Yaskawa INFORM job: SKRZYNIA_4940_0_STOPNI_1OBR.JBI

/JOB
//NAME SKRZYNIA_4940_0_STOPNI_1OBR
///FOLDERNAME 02-SKRZYNIE_JOBS
//POS
///NPOS 518,518,0,43,0,0
///TOOL 0
///POSTYPE PULSE
///PULSE
C00000=1055,-24125,84372,288,19725,204
C00001=1055,-24125,84372,288,19725,204
C00002=0,-15438,65714,0,-68532,0
C00003=25524,-25821,36823,19654,-58495,38520
C00004=23988,-24960,37134,18595,-57837,38812
C00005=22822,-23954,37534,17811,-57199,39017
C00006=22935,-24057,37491,17887,-57262,38997
C00007=20006,-24258,37408,15644,-56932,39751
C00008=24402,-25289,37013,18874,-58060,38740
C00009=22585,-24665,40358,17164,-59622,30036
C00010=23477,-23257,40205,18030,-58646,29630
C00011=22519,-22398,40568,17384,-58125,29795
C00012=22700,-22567,40495,17506,-58225,29764
C00013=19339,-22794,40398,14955,-57865,30607
C00014=24825,-24328,39798,18931,-59350,29401
C00015=0,-15438,65714,0,-68532,0
C00016=25524,-25821,36823,19654,-58495,38520
C00017=23988,-24960,37134,18595,-57837,38812
C00018=22822,-23954,37534,17811,-57199,39017
C00019=22935,-24057,37491,17887,-57262,38997
C00020=20006,-24258,37408,15644,-56932,39751
C00021=24402,-25289,37013,18874,-58060,38740
C00022=22585,-24665,40358,17164,-59622,30036
C00023=23477,-23257,40205,18030,-58646,29630
C00024=22519,-22398,40568,17384,-58125,29795
C00025=22700,-22567,40495,17506,-58225,29764
C00026=19339,-22794,40398,14955,-57865,30607
C00027=24825,-24328,39798,18931,-59350,29401
C00028=32755,-32613,25711,29640,-48730,33694
C00029=25632,-30899,26166,23992,-46203,35378
C00030=24264,-29862,26497,22996,-45413,35639
C00031=24403,-29974,26459,23097,-45496,35612
C00032=20575,-30233,26374,19602,-44891,36810
C00033=26556,-31526,25988,24663,-46720,35206
C00034=30467,-34548,18624,42252,-31099,25545
C00035=27667,-31817,21023,40298,-29340,25942
C00036=26226,-30681,21430,39338,-28403,26129
C00037=26403,-30829,21375,39455,-28520,26106
C00038=23300,-31093,21277,35654,-27590,27434
C00039=27667,-31817,21023,40298,-29340,25942
C00040=26028,-43665,26580,-39946,8682,24640
C00041=27956,-30595,53065,-101898,6609,54413
C00042=26028,-43663,26580,-39944,8677,24639
C00043=38124,-35330,25507,26155,-45940,34419
C00044=17528,-33021,25719,14295,-44761,40001
C00045=28412,-21339,35361,20830,-70681,36412
C00046=27333,-20260,35973,20228,-70115,36596
C00047=27560,-20497,35837,20355,-70235,36556
C00048=24830,-20816,35654,18694,-69859,37222
C00049=28877,-18893,40191,20941,-72149,36569
C00050=27817,-32566,25782,25532,-47502,36865
C00051=25779,-31294,26110,24054,-46400,37243
C00052=24344,-30243,26427,23007,-45578,37515
C00053=24432,-30312,26405,23072,-45630,37498
C00054=20021,-30599,26315,19050,-44944,38872
C00055=26262,-31616,26021,24405,-46667,37153
C00056=27439,-32346,25835,25259,-47302,36935
C00057=25659,-31170,26146,23974,-46312,37260
C00058=24581,-30384,26384,23190,-45695,37464
C00059=24689,-30466,26358,23269,-45758,37444
C00060=20001,-30771,26264,18999,-45026,38899
C00061=26308,-31607,26026,24448,-46671,37139
C00062=29920,-29398,24569,49034,-27892,27689
C00063=29115,-28721,24834,48649,-27358,27707
C00064=27674,-27540,25333,47889,-26423,27783
C00065=27794,-27645,25287,47952,-26502,27777
C00066=24751,-27949,25156,44290,-25406,29014
C00067=29115,-28721,24834,48649,-27358,27707
C00068=46709,-36638,22429,58955,-37174,26391
C00069=28781,-29734,22128,31822,13650,18140
C00070=28781,-29734,22128,31822,47214,18140
C00071=28781,-29734,22128,31822,47214,18140
C00072=54276,-43673,-470,62120,-47739,23626
C00073=41752,-40945,238,55421,-40682,25053
C00074=39867,-39951,547,54583,-39468,25162
C00075=39963,-40004,529,54625,-39531,25157
C00076=37168,-40414,400,52318,-38319,25966
C00077=43368,-42081,-2849,57747,-40820,23950
C00078=38095,-40136,7813,41252,-44156,24924
C00079=33231,-38681,8176,37792,-41757,25918
C00080=31538,-37640,8473,36716,-40716,26179
C00081=31687,-37737,8444,36811,-40809,26155
C00082=27389,-38154,8322,32773,-39589,27627
C00083=33834,-39023,8084,38175,-42120,25821
C00084=27585,-47842,-289,32095,-40789,28095
C00085=4801,-35772,25187,4593,-28023,-82032
C00086=17634,-23800,39238,9573,-31425,-73339
C00087=17634,-23800,39238,9573,-31425,-73339
C00088=16549,-22464,39800,8390,-30730,-72975
C00089=16684,-22641,39722,8536,-30818,-73021
C00090=16684,-19968,45512,8078,-32771,-72767
C00091=17634,-23800,39238,9573,-31425,-73339
C00092=17837,-21535,44509,9322,-33342,-73155
C00093=17837,-21535,44509,9322,-33342,-73155
C00094=16866,-20378,45014,8305,-32755,-72853
C00095=17032,-20588,44918,8481,-32857,-72905
C00096=17032,-17542,51480,8009,-35060,-72636
C00097=17837,-21535,44509,9322,-33342,-73155
C00098=-20829,-18800,50532,-12466,-37179,-77446
C00099=-19934,-17904,50946,-11618,-36715,-77676
C00100=-20044,-18019,50891,-11723,-36773,-77647
C00101=-20044,-15288,56753,-11218,-38713,-77950
C00102=-20966,-18928,50473,-12596,-37250,-77413
C00103=-20884,-26676,33664,-14451,-31668,-76336
C00104=-20884,-26676,33664,-14451,-31668,-76336
C00105=-19557,-25338,34176,-13080,-30873,-76751
C00106=-19691,-25483,34117,-13220,-30955,-76709
C00107=-19691,-22773,39998,-12506,-32911,-77106
C00108=-20642,-26447,33747,-14206,-31526,-76411
C00109=-33629,-40566,17444,-29603,-33447,-71192
C00110=-33629,-40566,17444,42578,-32312,-84654
C00111=-42160,-31266,16400,42578,-32312,-84654
C00112=-87798,-804,48829,-20188,-26072,-60966
C00113=-76454,-11934,10236,-25964,7954,-64922
C00114=-76448,-11928,10235,-25961,7944,-64914
C00115=-68643,-7759,-23318,-14097,50582,-74897
C00116=-70868,-8793,-8075,-29663,30364,-70765
C00117=-67243,-1968,12282,-49553,26687,-63567
C00118=-68655,-309,14069,-48513,25966,-64203
C00119=-67497,-1678,12591,-49367,26558,-63682
C00120=-71436,-723,2905,-26484,35140,-73726
C00121=-71436,176,6426,-27636,33595,-73066
C00122=-71434,778,8668,-28412,32633,-72624
C00123=-68624,-2689,-85,-28291,36551,-72622
C00124=-99375,3692,5712,40719,48607,-84097
C00125=-94964,4957,10918,40408,44640,-83792
C00126=-93063,6047,12199,39572,43744,-83178
C00127=-94964,4957,10918,40408,44640,-83792
C00128=-94964,5754,13918,41385,43553,-84439
C00129=-94964,4957,10918,40408,44640,-83792
C00130=-90271,-412,-5146,23417,46876,-76529
C00131=-83133,-4088,-8267,6704,41492,-71542
C00132=-83133,-4088,-8267,6704,41492,-71542
C00133=-83133,-4088,-8267,6704,41492,-11598
C00134=-83133,-16026,-8267,6704,41492,-11598
C00135=-83133,-16026,-8267,6704,41492,-11598
C00136=-48225,-19387,30619,3889,32460,-6728
C00137=56943,-39861,25115,1795,-37402,-69601
C00138=29960,-38386,-19607,-115769,-41858,-24264
C00139=65721,-6478,18155,-133323,-22195,3361
C00140=70544,4411,32968,-134868,-18623,4660
C00141=71874,8263,38598,-134556,-17327,4659
C00142=72629,9390,40002,-135279,-16924,5107
C00143=71441,7638,37831,-134139,-17555,4406
C00144=77146,8888,25050,-166574,-32612,18372
C00145=77146,10029,28643,-166204,-31014,18167
C00146=77146,11198,32202,-165803,-29459,17947
C00147=75508,4678,16951,-165715,-35157,17778
C00148=68680,12216,24468,-164340,-40455,-13359
C00149=68362,12845,25743,-164045,-40097,-13561
C00150=68362,13700,28585,-163752,-38808,-13742
C00151=68362,12845,25743,-164045,-40097,-13561
C00152=64993,-1168,28876,-102971,-10760,-49875
C00153=63888,481,30670,-102324,-11438,-50313
C00154=64993,-1168,28876,-102971,-10760,-49875
C00155=58588,-14653,4620,-120782,-19611,-35794
C00156=29960,-38386,-19607,-115769,-41858,-24264
C00157=56943,-39861,25115,1795,-37402,-69601
C00158=-1002,-39861,25115,1795,-37402,-69601
C00159=-1001,-39858,25114,1795,-37402,0
C00160=6591,-33902,35532,5956,-1761,-1932
C00161=6592,-33900,35531,103508,-35512,-26314
C00162=-99253,-13690,44082,59847,13407,-31313
C00163=-85045,-36869,-4353,28502,-22832,-52282
C00164=-92346,-18713,13565,21110,-22545,-55257
C00165=-85732,-21202,11427,30682,-24763,-59235
C00166=-84559,-15616,15722,33768,-24118,-60665
C00167=-84150,-13282,17685,34842,-23935,-61163
C00168=-83260,-12880,18034,36130,-24218,-61709
C00169=-84150,-13282,17685,34842,-23935,-61163
C00170=-85365,-11775,19006,33430,-23307,-60600
C00171=-84150,-13282,17685,34842,-23935,-61163
C00172=-85786,-16909,14677,31743,-23900,-59790
C00173=-84150,-13282,17685,34842,-23935,-61163
C00174=-83215,-12861,18051,36194,-24233,-61735
C00175=-84150,-13282,17685,34842,-23935,-61163
C00176=-85327,-11825,18959,33476,-23327,-60618
C00177=-84150,-13282,17685,34842,-23935,-61163
C00178=-87841,-18519,13420,28367,-23534,-58339
C00179=-84150,-13282,17685,34842,-23935,-61163
C00180=-83292,-12894,18020,36083,-24208,-61688
C00181=-84150,-13282,17685,34842,-23935,-61163
C00182=-85185,-12008,18799,33646,-23400,-60687
C00183=-84150,-13282,17685,34842,-23935,-61163
C00184=-86371,-18277,13606,30568,-23951,-59265
C00185=-84345,-13370,17612,34554,-23873,-61041
C00186=-83240,-12871,18042,36158,-24225,-61720
C00187=-84345,-13370,17612,34554,-23873,-61041
C00188=-85365,-12110,18711,33368,-23345,-60568
C00189=-84345,-13370,17612,34554,-23873,-61041
C00190=-86191,-19647,12567,30467,-24278,-59187
C00191=-84345,-13372,17610,34552,-23873,-61039
C00192=-83096,-12807,18098,36363,-24268,-61804
C00193=-84345,-13372,17610,34552,-23873,-61039
C00194=-85268,-12232,18600,33480,-23393,-60612
C00195=-84345,-13372,17610,34552,-23873,-61039
C00196=-84814,-16043,15376,33312,-24093,-60464
C00197=-84104,-13265,17702,34906,-23948,-61189
C00198=-82960,-12743,18153,36555,-24313,-61887
C00199=-84104,-13265,17702,34906,-23948,-61189
C00200=-84979,-12194,18635,33901,-23496,-60788
C00201=-84104,-13265,17702,34906,-23948,-61189
C00202=-86610,-16845,14732,30573,-23614,-59301
C00203=-84104,-13265,17702,34906,-23948,-61189
C00204=-82793,-12667,18222,36790,-24370,-61986
C00205=-84104,-13265,17702,34906,-23948,-61189
C00206=-84888,-12305,18537,34004,-23540,-60830
C00207=-84104,-13265,17702,34906,-23948,-61189
C00208=-83806,-19585,12613,33764,-25080,-60559
C00209=-83675,-13072,17868,35530,-24083,-61453
C00210=-82553,-12556,18319,37130,-24451,-62127
C00211=-83675,-13072,17868,35530,-24083,-61453
C00212=-84378,-12223,18610,34735,-23716,-61138
C00213=-83675,-13072,17868,35530,-24083,-61453
C00214=-87149,-17993,13826,29513,-23647,-58830
C00215=-84104,-13265,17702,34906,-23948,-61189
C00216=-82640,-12594,18285,37014,-24425,-62079
C00217=-84104,-13265,17702,34906,-23948,-61189
C00218=-84792,-12429,18430,34119,-23592,-60877
C00219=-84104,-13265,17702,34906,-23948,-61189
C00220=-83583,-9185,30892,23668,-36042,-57025
C00221=-85789,-8328,35795,20592,-37093,-55378
C00222=-85786,-16735,14816,31782,-23869,-59812
C00223=-84103,-13263,17702,34906,-23947,-61191
C00224=-83225,-12865,18046,36177,-24227,-61729
C00225=-84103,-13263,17702,34906,-23947,-61191
C00226=-84774,-12447,18412,34138,-23599,-60886
C00227=-84103,-13263,17702,34906,-23947,-61191
C00228=-86149,-16246,6730,18897,-35239,-57128
C00229=-86244,-15289,7532,18875,-35060,-57127
C00230=-85361,-14893,7870,19824,-35193,-57574
C00231=-86244,-15289,7532,18875,-35060,-57127
C00232=-86889,-14409,8282,18264,-34784,-56850
C00233=-86244,-15289,7532,18875,-35060,-57127
C00234=-90262,-21765,2389,14114,-35574,-54847
C00235=-90262,-21765,2389,28730,-17672,-54847
C00236=-89967,-19086,25635,28730,-17672,-54847
C00237=568,-24029,84339,168,19981,112
C00238=568,-24677,83015,164,20405,113
C00239=101153,-24598,83176,165,20353,113
C00240=101153,-24598,83176,165,20353,113
C00241=89967,-19086,25635,-28730,-17672,54847
C00242=90262,-21765,2389,-28730,-17672,54847
C00243=86932,-18662,4771,-17876,-35519,56628
C00244=86578,-15436,7408,-18515,-35011,56957
C00245=85428,-14922,7844,-19753,-35183,57541
C00246=84405,-14447,8250,-20842,-35348,58054
C00247=85428,-14922,7844,-19753,-35183,57541
C00248=86134,-13973,8661,-19091,-34881,57237
C00249=85428,-14922,7844,-19753,-35183,57541
C00250=85786,-16735,14816,-31782,-23869,59812
C00251=83514,-12996,17929,-35760,-24132,61552
C00252=82296,-12429,18424,-37488,-24534,62281
C00253=83514,-12996,17929,-35760,-24132,61552
C00254=84266,-12085,18725,-34910,-23738,61214
C00255=83514,-12996,17929,-35760,-24132,61552
C00256=87323,-6914,39851,-18853,-38149,44508
C00257=83118,-12818,18089,-36330,-24263,61791
C00258=81969,-12276,18566,-37944,-24648,62472
C00259=83118,-12818,18089,-36330,-24263,61791
C00260=83927,-11846,18941,-35423,-23842,61433
C00261=83118,-12818,18089,-36330,-24263,61791
C00262=83806,-19585,12613,-33764,-25080,60559
C00263=83148,-12832,18077,-36287,-24254,61773
C00264=81889,-12236,18598,-38058,-24676,62520
C00265=83148,-12832,18077,-36287,-24254,61773
C00266=83900,-11930,18867,-35446,-23862,61440
C00267=83148,-12832,18077,-36287,-24254,61773
C00268=86610,-16845,14732,-30573,-23614,59301
C00269=82493,-13239,17725,-37070,-24559,62089
C00270=81442,-12739,18159,-38529,-24915,62703
C00271=82493,-13239,17725,-37070,-24559,62089
C00272=83435,-12133,18689,-36040,-24063,61682
C00273=82493,-13239,17725,-37070,-24559,62089
C00274=84814,-16043,15376,-33312,-24093,60464
C00275=82555,-13613,17404,-36910,-24580,62015
C00276=81369,-13053,17885,-38558,-24979,62709
C00277=82555,-13613,17404,-36910,-24580,62015
C00278=83568,-12431,18429,-35805,-24046,61580
C00279=82555,-13613,17404,-36910,-24580,62015
C00280=86191,-19647,12567,-30467,-24278,59187
C00281=82500,-13648,17375,-36975,-24607,62039
C00282=81594,-13224,17740,-38236,-24911,62571
C00283=82500,-13648,17375,-36975,-24607,62039
C00284=83449,-12543,18332,-35941,-24104,61633
C00285=82500,-13648,17375,-36975,-24607,62039
C00286=86371,-18277,13606,-30568,-23951,59265
C00287=82904,-13790,17251,-36416,-24470,61808
C00288=81796,-13275,17692,-37971,-24838,62464
C00289=82904,-13790,17251,-36416,-24470,61808
C00290=83696,-12867,18046,-35547,-24051,61466
C00291=82904,-13790,17251,-36416,-24470,61808
C00292=87841,-18519,13420,-28367,-23534,58339
C00293=82748,-13879,17174,-36603,-24542,61883
C00294=81789,-13434,17554,-37946,-24861,62449
C00295=82748,-13879,17174,-36603,-24542,61883
C00296=83603,-12888,18026,-35668,-24086,61514
C00297=82748,-13879,17174,-36603,-24542,61883
C00298=85786,-16909,14677,-31743,-23900,59790
C00299=82339,-14116,16972,-37087,-24733,62079
C00300=81557,-13752,17280,-38171,-24994,62536
C00301=82339,-14116,16972,-37087,-24733,62079
C00302=83390,-12909,18006,-35951,-24172,61633
C00303=82339,-14116,16972,-37087,-24733,62079
C00304=85732,-21202,11427,-30682,-24763,59235
C00305=82398,-14365,16763,-36952,-24745,62014
C00306=81340,-13876,17176,-38416,-25096,62632
C00307=82398,-14365,16763,-36952,-24745,62014
C00308=83629,-12951,17972,-35620,-24090,61491
C00309=82398,-14365,16763,-36952,-24745,62014
C00310=83775,-36460,5778,-32556,-23750,56951
C00311=69856,-53931,-13446,-33557,-28911,29591
C00312=0,-24029,84339,0,19981,0
C00313=0,-24029,84339,0,19981,0
C00314=0,-52280,40443,0,6876,0
C00315=43695,-41610,22646,45477,-37580,9181
C00316=79833,-32060,29151,65065,-75499,17030
C00317=46589,-23543,32575,47437,-59456,19719
C00318=34746,-28644,20980,31794,-60034,26371
C00319=20694,-31959,9398,15734,-60691,34314
C00320=58029,-25484,23838,55879,-68285,17494
C00321=64424,-28491,31029,58630,-66351,17656
C00322=0,-52280,40443,0,6876,0
C00323=0,-52280,40443,0,6876,0
C00324=23755,-47704,18289,26329,-25233,13971
C00325=32804,-46073,6525,41905,-31120,14425
C00326=62562,-39100,6547,70046,-55853,12125
C00327=48126,-33841,8393,64372,-47199,12361
C00328=31253,-44096,-7366,36514,-42480,22085
C00329=59828,-44646,-5405,72855,-48572,12139
C00330=0,-38761,66314,0,-763,0
C00331=0,-44757,54667,0,2744,0
C00332=40382,-38226,12225,48505,-40693,16039
C00333=55481,-27484,23768,62968,-54833,11978
C00334=49931,-26522,24223,59987,-51967,12537
C00335=41382,-34078,10932,46059,-50502,16311
C00336=55330,-33748,11238,57660,-59334,12681
C00337=78664,-24436,10378,82837,-79111,12029
C00338=75189,-23065,11287,81851,-76948,11927
C00339=75189,-45249,11287,81851,-38847,11927
C00340=29880,-45249,11287,43145,-11324,11927
C00341=0,-24029,84339,0,19981,0
C00342=0,-24026,84338,1,19977,2
C00343=4264,-34194,25387,4006,-26954,-29436
C00344=4264,-34194,25387,4006,-26954,-81856
C00345=-21478,-27798,32214,-15234,-31599,-76056
C00346=-19679,-23059,39354,-12567,-32689,-77067
C00347=16724,-20576,44291,8212,-32395,-72836
C00348=21329,-26386,39716,13285,-34016,-74401
C00349=-23778,-26243,38799,-16502,-35132,-75964
C00350=-20075,-15782,55752,-11329,-38404,-77896
C00351=16874,-17447,51356,7863,-34895,-72604
C00352=18580,-28601,30698,11472,-29284,-74138
C00353=6126,-41331,18955,6697,-26557,-30383
C00354=1,-24024,84337,2,19973,1
C00355=-64243,-26178,31107,-39513,40312,-5844
C00356=-72148,3973,56008,-35470,42045,-10522
C00357=-72090,16396,76301,-42067,35650,-6519
C00358=-69388,15725,61378,-31740,35177,-8719
C00359=-69127,27099,75569,-32744,34250,-8088
C00360=-67573,2495,11285,-21767,57629,-15193
C00361=-77819,19629,29798,-10454,63174,-20704
C00362=-72990,23583,14304,-10735,77209,-20379
C00363=-74593,38003,46707,-11043,65751,-19814
C00364=-73236,38943,48295,-11400,65557,-19316
C00365=-73329,42107,51779,-6346,67443,-19636
C00366=-87142,34654,46174,17622,63862,-25393
C00367=-87240,36727,48611,18897,66604,-25032
C00368=-99033,21517,12213,24947,79702,-26203
C00369=-91500,-14196,-34781,24472,81625,-22832
C00370=-100472,-45007,-27818,8167,67201,-29302
C00371=0,-36642,16905,0,48372,0
C00372=66009,-61997,-62105,21406,63483,18379
C00373=97242,-23579,-39442,10179,68876,30321
C00374=73684,-7073,-17511,24638,68131,29022
C00375=59136,7235,6676,33270,66602,27507
C00376=54816,14937,6234,39741,69494,31070
C00377=54365,20668,19279,41017,66202,29418
C00378=64503,4223,2857,29650,48528,26647
C00379=75622,3202,-3149,3890,49494,34281
C00380=88036,13177,2413,-18568,66573,35876
C00381=90462,21593,10123,-22613,76266,34479
C00382=92450,29224,20002,-25750,81642,33727
C00383=94949,8131,-12163,-20291,74229,36861
C00384=94949,8084,-13484,-20215,75047,36712
C00385=70412,-34016,-52305,-11724,65624,29757
C00386=44268,-30306,-1568,-7370,48673,18708
C00387=1,-24024,84337,2,19973,1
C00388=1,-24024,84337,2,19973,1
C00389=3796,-57671,22373,2336,-25309,-753
C00390=52632,-34554,16626,51161,-63050,5622
C00391=41454,-25301,37199,36495,-58855,24340
C00392=36675,-26014,30916,36565,-54296,30358
C00393=31298,-42259,-4306,53964,-29254,17939
C00394=62932,-33588,12189,66848,-61063,18031
C00395=57521,-31202,17284,65112,-55174,10876
C00396=49869,-26949,23557,59706,-52171,12606
C00397=49645,-31441,12217,55064,-56016,13120
C00398=55330,-33748,11238,57660,-59334,12681
C00399=29694,-28537,50295,31543,-18263,8508
C00400=1,-24024,84337,2,19973,1
C00401=1,-24024,84337,2,19973,1
C00402=57188,-41777,19973,48132,-58706,4905
C00403=55566,-48748,-16991,79805,-45048,-6941
C00404=49908,-48716,-25784,90749,-41340,-3650
C00405=34097,-50090,-26426,85195,-27377,-3312
C00406=29342,-53468,-37504,108423,-23986,-15312
C00407=55456,-69347,-61742,105381,-46819,-11205
C00408=12119,-24859,71505,13236,4440,2633
C00409=-91085,-34291,10385,1908,-24348,-42097
C00410=-86191,-19647,12567,30467,-24278,-59187
C00411=-99336,-11722,19052,-14323,-20229,-40037
C00412=-98356,-11562,19564,-10422,-20330,-41507
C00413=-99474,-20389,12397,-11593,-22150,-41069
C00414=0,-52280,40443,0,6876,0
C00415=98750,-34911,19055,13387,-20552,33529
C00416=85481,-22689,10385,-30594,-25183,59147
C00417=97204,-12655,18233,8807,-19987,42423
C00418=97248,-12883,18033,8874,-20029,42393
C00419=96230,-24528,9149,6144,-22576,43630
C00420=0,-52280,40443,0,6876,0
C00421=0,-52280,40443,0,6876,0
C00422=-90140,-60305,18108,-2708,1721,-7625
C00423=-95594,-27428,6866,-4663,-19832,-42154
C00424=-99356,-13410,18355,-15385,-17730,-37479
C00425=-99591,-10931,20459,-16242,-17374,-37088
C00426=-99412,-10883,20509,-15863,-17339,-37249
C00427=-100555,-16348,15834,-17428,-18409,-36628
C00428=-90140,-60305,18108,-2708,1721,-7625
C00429=0,-52280,40443,0,6876,0
C00430=84259,-57935,27522,-3761,3673,6310
C00431=86507,-39672,4297,-27618,-16640,46340
C00432=79502,-31038,5321,-35142,-29552,60614
C00433=87509,-17632,14108,-29072,-23467,58651
C00434=100494,-12641,18246,19637,-20925,37756
C00435=99867,-15453,10402,24266,-14765,33998
C00436=100699,-20865,6123,24471,-16015,33991
C00437=86507,-39672,4297,-27618,-16640,46340
C00438=84259,-57935,27522,-3761,3673,6310
C00439=0,-52280,40443,0,6876,0
C00440=0,-27933,77061,0,20812,0
C00441=0,-27933,77061,0,20812,0
C00442=0,-52280,40443,0,6876,0
C00443=-91970,-60791,14435,-3343,512,-9412
C00444=-99196,-15868,16098,-13748,-19297,-38710
C00445=-99196,-15868,16098,-13748,-19297,-38710
C00446=-99196,-15868,16098,-13748,-19297,-38710
C00447=-85896,-11794,19566,31613,-21074,-58206
C00448=-87494,-11929,19445,26784,-20178,-56163
C00449=-99562,-16264,15781,-14410,-19427,-38431
C00450=-99196,-15868,16098,-13748,-19297,-38710
C00451=-91970,-60791,14435,-3343,512,-9412
C00452=0,-52280,40443,0,6876,0
C00453=91083,-60784,14823,-9043,-825,15173
C00454=83869,-19403,12921,-33769,-24740,60260
C00455=83869,-19403,12921,-33769,-24740,60260
C00456=83420,-14897,16486,-35538,-24144,61113
C00457=90681,-11839,19658,-13770,-20778,51433
C00458=90505,-11641,19895,-14005,-20849,51502
C00459=95871,-14889,15992,4901,-19605,43825
C00460=83869,-19403,12921,-33769,-24740,60260
C00461=91083,-60784,14823,-9043,-825,15173
C00462=0,-52280,40443,0,6876,0
C00463=-91526,-60598,16699,7584,176,-13289
C00464=-94392,-6553,48683,5805,-47321,-49764
C00465=-88951,-345,54953,10686,-47392,-51569
C00466=-88305,5764,62037,11205,-47732,-51744
C00467=-91201,-14114,9416,8552,-34389,-51801
C00468=-84917,-15593,15742,33275,-23984,-60461
C00469=-81669,-15982,15425,37506,-25258,-62202
C00470=-79867,-25377,9541,37586,-25936,-59971
C00471=-91415,-60262,16631,7870,-73,-13734
C00472=24,-24029,84339,7,19981,5
C00473=160,-24029,84339,47,19981,32
C00474=99096,-24029,84339,47,19981,32
C00475=99096,-24029,84339,47,19981,32
C00476=89967,-19086,25635,-28730,-17672,54847
C00477=85786,-16735,14816,-31782,-23869,59812
C00478=83492,-14473,16674,-35480,-24338,61406
C00479=82747,-11488,19289,-37317,-24361,62210
C00480=85506,-13730,8787,-19466,-34817,57474
C00481=85505,-16299,6686,-19564,-35388,57437
C00482=89967,-19086,25635,-28730,-17672,54847
C00483=568,-24029,84339,168,19981,112
C00484=568,-24029,84339,168,19981,112
C00485=-91970,-60791,14435,-3343,512,-9412
C00486=-86948,-23217,10819,28314,-23349,-56438
C00487=-85895,-16522,15767,31843,-22281,-58087
C00488=-93744,1669,52928,2829,-38206,-34736
C00489=-93484,-766,47198,3260,-36104,-34933
C00490=-86145,-24679,9854,29028,-23971,-56682
C00491=-100471,-58311,4157,14142,-4822,-27614
C00492=-68517,-58311,4157,14142,-4822,-27614
C00493=0,-52280,40443,0,6876,0
C00494=91083,-60784,14823,-9043,-825,15173
C00495=83869,-19403,12921,-33769,-24740,60260
C00496=82620,-18743,14708,-32942,-26226,58979
C00497=84031,-4887,35984,-19530,-40379,54984
C00498=84316,-7987,27276,-19995,-38113,55712
C00499=84798,-22668,11879,-29033,-26372,57255
C00500=91083,-60784,14823,-9043,-825,15173
C00501=0,-52280,40443,0,6876,0
C00502=-6369,-39206,65423,-4801,-482,2563
C00503=-97287,-29142,12714,-8673,-22288,-37832
C00504=-86191,-19647,12567,30467,-24278,-59187
C00505=-85671,-16302,15857,30808,-24404,-58999
C00506=-100216,-10426,22391,-15020,-22581,-38655
C00507=-96259,-10424,22189,-2878,-17380,-43087
C00508=-87910,-17792,15835,25414,-24996,-56048
C00509=-97287,-29142,12714,-8673,-22288,-37832
C00510=0,-52280,40443,0,6876,0
C00511=92301,-25634,22749,2368,-15645,37646
C00512=83738,-18329,13570,-34202,-24868,60772
C00513=90255,-12942,18284,-15153,-20833,52586
C00514=93508,-13158,18002,-4292,-20124,47959
C00515=80226,-20465,12178,-39626,-27411,62762
C00516=92301,-25634,22749,2368,-15645,37646
C00517=0,-52280,40443,0,6876,0
BC00000=413138
BC00001=413138
BC00002=413138
BC00003=290246
BC00004=290246
BC00005=290246
BC00006=290246
BC00007=290246
BC00008=290246
BC00009=347127
BC00010=347132
BC00011=347132
BC00012=347132
BC00013=347132
BC00014=347132
BC00015=413138
BC00016=413134
BC00017=413134
BC00018=413134
BC00019=413134
BC00020=413134
BC00021=413134
BC00022=474623
BC00023=474628
BC00024=474628
BC00025=474628
BC00026=474628
BC00027=474628
BC00028=522849
BC00029=522849
BC00030=522849
BC00031=522849
BC00032=522849
BC00033=522849
BC00034=550624
BC00035=553627
BC00036=553627
BC00037=553627
BC00038=553627
BC00039=553627
BC00040=470246
BC00041=618860
BC00042=673957
BC00043=691345
BC00044=686969
BC00045=712250
BC00046=712250
BC00047=712250
BC00048=712250
BC00049=712250
BC00050=708270
BC00051=708270
BC00052=708270
BC00053=708270
BC00054=708270
BC00055=708270
BC00056=770184
BC00057=770184
BC00058=770184
BC00059=770184
BC00060=770184
BC00061=770184
BC00062=788736
BC00063=788736
BC00064=788736
BC00065=788736
BC00066=788736
BC00067=788736
BC00068=729895
BC00069=703565
BC00070=703565
BC00071=802913
BC00072=891475
BC00073=891475
BC00074=891475
BC00075=891475
BC00076=891475
BC00077=891475
BC00078=934475
BC00079=934475
BC00080=934475
BC00081=934475
BC00082=934475
BC00083=934475
BC00084=934475
BC00085=880430
BC00086=895791
BC00087=895791
BC00088=895791
BC00089=895791
BC00090=895791
BC00091=895791
BC00092=900237
BC00093=900237
BC00094=900237
BC00095=900237
BC00096=900237
BC00097=900237
BC00098=900237
BC00099=900237
BC00100=900237
BC00101=900237
BC00102=900237
BC00103=900237
BC00104=900237
BC00105=900237
BC00106=900237
BC00107=900237
BC00108=900237
BC00109=900237
BC00110=900237
BC00111=900237
BC00112=900237
BC00113=900237
BC00114=917989
BC00115=929075
BC00116=945779
BC00117=945779
BC00118=945779
BC00119=945779
BC00120=945779
BC00121=945779
BC00122=945780
BC00123=945780
BC00124=945780
BC00125=945780
BC00126=945780
BC00127=945780
BC00128=945780
BC00129=945780
BC00130=936157
BC00131=921523
BC00132=896258
BC00133=896258
BC00134=896258
BC00135=863076
BC00136=828643
BC00137=900237
BC00138=900237
BC00139=900237
BC00140=916451
BC00141=921612
BC00142=921612
BC00143=921612
BC00144=921612
BC00145=921612
BC00146=921612
BC00147=921612
BC00148=921612
BC00149=921612
BC00150=921612
BC00151=921612
BC00152=921612
BC00153=921612
BC00154=921612
BC00155=916099
BC00156=869515
BC00157=838793
BC00158=838793
BC00159=854156
BC00160=785093
BC00161=785096
BC00162=785096
BC00163=854699
BC00164=886829
BC00165=902188
BC00166=902188
BC00167=902188
BC00168=902188
BC00169=902188
BC00170=902188
BC00171=902188
BC00172=840744
BC00173=840744
BC00174=840744
BC00175=840744
BC00176=840744
BC00177=840744
BC00178=779300
BC00179=779300
BC00180=779300
BC00181=779300
BC00182=779300
BC00183=779300
BC00184=717855
BC00185=717855
BC00186=717855
BC00187=717855
BC00188=717855
BC00189=717855
BC00190=656405
BC00191=656405
BC00192=656405
BC00193=656405
BC00194=656405
BC00195=656405
BC00196=594961
BC00197=594961
BC00198=594961
BC00199=594961
BC00200=594961
BC00201=594961
BC00202=533517
BC00203=533517
BC00204=533517
BC00205=533517
BC00206=533517
BC00207=533517
BC00208=472073
BC00209=472073
BC00210=472073
BC00211=472073
BC00212=472073
BC00213=472073
BC00214=410629
BC00215=410629
BC00216=410629
BC00217=410629
BC00218=410629
BC00219=410629
BC00220=410629
BC00221=349186
BC00222=349186
BC00223=349186
BC00224=349186
BC00225=349186
BC00226=349186
BC00227=349186
BC00228=336469
BC00229=336469
BC00230=336469
BC00231=336469
BC00232=336469
BC00233=336469
BC00234=336469
BC00235=336469
BC00236=336469
BC00237=336469
BC00238=511557
BC00239=512005
BC00240=363797
BC00241=336469
BC00242=336469
BC00243=337415
BC00244=337415
BC00245=337415
BC00246=337415
BC00247=337415
BC00248=337415
BC00249=337415
BC00250=349186
BC00251=350137
BC00252=350137
BC00253=350137
BC00254=350137
BC00255=350137
BC00256=410629
BC00257=411580
BC00258=411580
BC00259=411580
BC00260=411580
BC00261=411580
BC00262=472073
BC00263=473025
BC00264=473025
BC00265=473025
BC00266=473025
BC00267=473025
BC00268=533517
BC00269=534468
BC00270=534468
BC00271=534468
BC00272=534468
BC00273=534468
BC00274=594961
BC00275=594961
BC00276=594961
BC00277=594961
BC00278=594961
BC00279=594961
BC00280=656405
BC00281=657350
BC00282=657350
BC00283=657350
BC00284=657350
BC00285=657350
BC00286=717855
BC00287=718799
BC00288=718799
BC00289=718799
BC00290=718799
BC00291=718799
BC00292=779300
BC00293=780245
BC00294=780245
BC00295=780245
BC00296=780245
BC00297=780245
BC00298=840744
BC00299=841691
BC00300=841691
BC00301=841691
BC00302=841691
BC00303=841691
BC00304=902188
BC00305=903136
BC00306=903136
BC00307=903136
BC00308=903136
BC00309=903136
BC00310=866428
BC00311=742376
BC00312=673191
BC00313=769966
BC00314=716865
BC00315=723595
BC00316=717171
BC00317=717171
BC00318=716481
BC00319=715784
BC00320=716000
BC00321=727625
BC00322=716865
BC00323=820009
BC00324=882789
BC00325=908954
BC00326=917484
BC00327=934308
BC00328=923719
BC00329=887066
BC00330=801718
BC00331=499733
BC00332=475338
BC00333=456696
BC00334=456696
BC00335=417276
BC00336=417276
BC00337=493986
BC00338=514306
BC00339=485368
BC00340=478024
BC00341=473587
BC00342=774064
BC00343=862181
BC00344=867397
BC00345=900237
BC00346=900237
BC00347=895790
BC00348=890024
BC00349=885535
BC00350=900237
BC00351=900237
BC00352=899465
BC00353=903057
BC00354=750918
BC00355=766280
BC00356=766280
BC00357=822990
BC00358=842876
BC00359=867815
BC00360=899747
BC00361=899747
BC00362=927256
BC00363=927256
BC00364=927256
BC00365=927257
BC00366=927257
BC00367=927258
BC00368=927258
BC00369=927258
BC00370=841916
BC00371=800514
BC00372=884054
BC00373=923174
BC00374=923175
BC00375=923175
BC00376=953422
BC00377=953422
BC00378=953422
BC00379=953422
BC00380=953422
BC00381=953425
BC00382=953425
BC00383=953425
BC00384=927019
BC00385=927019
BC00386=858206
BC00387=735557
BC00388=469153
BC00389=499904
BC00390=541592
BC00391=531564
BC00392=529848
BC00393=579756
BC00394=529848
BC00395=333808
BC00396=332068
BC00397=295166
BC00398=294388
BC00399=454783
BC00400=441730
BC00401=632615
BC00402=778314
BC00403=778312
BC00404=778312
BC00405=778312
BC00406=835726
BC00407=836556
BC00408=566410
BC00409=707357
BC00410=656405
BC00411=656405
BC00412=717855
BC00413=717855
BC00414=680147
BC00415=662303
BC00416=657350
BC00417=657350
BC00418=718803
BC00419=718803
BC00420=683493
BC00421=792672
BC00422=792672
BC00423=896850
BC00424=895720
BC00425=895720
BC00426=925351
BC00427=927080
BC00428=792672
BC00429=792672
BC00430=792672
BC00431=887446
BC00432=903126
BC00433=903126
BC00434=903126
BC00435=936389
BC00436=936389
BC00437=887446
BC00438=792672
BC00439=792672
BC00440=700249
BC00441=546214
BC00442=546214
BC00443=546211
BC00444=546211
BC00445=406776
BC00446=406776
BC00447=406778
BC00448=468200
BC00449=468200
BC00450=546211
BC00451=546211
BC00452=546214
BC00453=546214
BC00454=507604
BC00455=410782
BC00456=410782
BC00457=410782
BC00458=472720
BC00459=472720
BC00460=507604
BC00461=546214
BC00462=546214
BC00463=516757
BC00464=383716
BC00465=349186
BC00466=349186
BC00467=336469
BC00468=349186
BC00469=410629
BC00470=416512
BC00471=515801
BC00472=520018
BC00473=474013
BC00474=474013
BC00475=403108
BC00476=336469
BC00477=349186
BC00478=349186
BC00479=349186
BC00480=337415
BC00481=337415
BC00482=336469
BC00483=336469
BC00484=428401
BC00485=546211
BC00486=591088
BC00487=591088
BC00488=591088
BC00489=531116
BC00490=529640
BC00491=529640
BC00492=529640
BC00493=529640
BC00494=546214
BC00495=589919
BC00496=595627
BC00497=609761
BC00498=555903
BC00499=534177
BC00500=546214
BC00501=529640
BC00502=651195
BC00503=765890
BC00504=777968
BC00505=778453
BC00506=779252
BC00507=832733
BC00508=840748
BC00509=730002
BC00510=671551
BC00511=714120
BC00512=780224
BC00513=780222
BC00514=841743
BC00515=841743
BC00516=741100
BC00517=660586
///POSTYPE BASE
///RECTAN
///RCONF 1,0,0,0,0,0,0,0,0,0,0,0,0,0,0,0,0,0,0,0,0,0,0,0
P00006=0.000,0.000,0.000,0.0000,0.0000,0.0000
///RCONF 0,0,0,0,0,0,0,0,0,0,0,0,0,0,0,0,0,0,0,0,0,0,0,0
P00021=6.550,-0.003,-5.735,0.0000,0.0000,0.0000
P00022=5.943,-0.018,-6.388,0.0000,0.0000,0.0000
P00023=7.025,-0.019,-7.168,0.0000,0.0000,0.0000
P00024=5.926,-0.047,-4.777,0.0000,0.0000,0.0000
///RCONF 1,0,0,0,0,0,0,0,0,0,0,0,0,0,0,0,0,0,0,0,0,0,0,0
P00098=-0.089,-2.467,4.059,0.0000,0.0000,0.0000
P00099=0.011,-2.380,1.226,0.0000,0.0000,0.0000
P00100=-0.081,2.558,4.482,0.0000,0.0000,0.0000
P00101=0.030,-2.286,2.993,0.0000,0.0000,0.0000
P00102=-0.005,-1.108,1.644,0.0000,0.0000,0.0000
P00103=-0.094,-3.400,4.200,0.0000,0.0000,0.0000
P00104=0.043,-2.127,5.826,0.0000,0.0000,0.0000
P00105=-0.043,0.662,5.286,0.0000,0.0000,0.0000
P00106=-0.018,-2.519,0.237,0.0000,0.0000,0.0000
P00107=-0.008,-4.537,-4.500,0.0000,0.0000,0.0000
P00108=0.014,-3.040,2.637,0.0000,0.0000,0.0000
P00109=0.017,-3.622,2.341,0.0000,0.0000,0.0000
///RCONF 0,0,0,0,0,0,0,0,0,0,0,0,0,0,0,0,0,0,0,0,0,0,0,0
P00280=-0.761,-1.221,0.004,0.0000,0.0000,0.0000
///RCONF 1,0,0,0,0,0,0,0,0,0,0,0,0,0,0,0,0,0,0,0,0,0,0,0
P00281=-0.866,-3.587,-0.008,0.0000,0.0000,0.0000
///RCONF 0,0,0,0,1,0,0,0,0,0,0,0,0,0,0,0,0,0,0,0,0,0,0,0
P00290=-0.023,-0.050,5.560,0.0000,0.0000,0.0000
///RCONF 1,0,0,0,0,0,0,0,0,0,0,0,0,0,0,0,0,0,0,0,0,0,0,0
P00291=0.002,-0.893,4.526,0.0000,0.0000,0.0000
P00301=0.046,-2.112,7.779,0.0000,0.0000,0.0000
P00302=-0.180,-2.409,6.326,0.0000,0.0000,0.0000
///RCONF 0,0,0,0,0,0,0,0,0,0,0,0,0,0,0,0,0,0,0,0,0,0,0,0
P00303=-0.004,-1.437,-4.584,0.0000,0.0000,0.0000
P00304=0.028,-1.666,-4.234,0.0000,0.0000,0.0000
P00305=-0.003,-1.920,-3.501,0.0000,0.0000,0.0000
P00306=0.015,-2.252,-3.054,0.0000,0.0000,0.0000
P00307=0.019,-2.151,-5.077,0.0000,0.0000,0.0000
P00308=-0.003,-2.092,-4.888,0.0000,0.0000,0.0000
P00309=-0.040,-2.205,-4.992,0.0000,0.0000,0.0000
P00310=-0.006,-2.490,-5.925,0.0000,0.0000,0.0000
P00311=-0.007,-2.079,-5.307,0.0000,0.0000,0.0000
P00350=11.519,-0.008,1.149,0.0000,0.0000,0.0000
P00351=13.563,-0.027,-0.653,0.0000,0.0000,0.0000
P00352=13.252,-0.027,-0.827,0.0000,0.0000,0.0000
P00353=10.971,-0.082,0.776,0.0000,0.0000,0.0000
P00354=-0.024,2.508,-1.824,0.0000,0.0000,0.0000
P00355=-0.001,2.528,-1.131,0.0000,0.0000,0.0000
P00356=-0.034,2.921,-0.262,0.0000,0.0000,0.0000
P00357=0.003,3.386,-0.091,0.0000,0.0000,0.0000
P00358=0.014,3.037,-0.020,0.0000,0.0000,0.0000
P00359=-0.005,2.731,0.912,0.0000,0.0000,0.0000
P00360=-0.011,3.412,0.438,0.0000,0.0000,0.0000
//INST
///DATE 2025/02/17 15:04
///ATTR SC,RW
///GROUP1 RB1,BS1
NOP
CALL JOB:MOVE_INTO_TUNNEL
MOVJ C00000 BC00000 VJ=30.00
'------------------------
'------------------------
'SPOINA SRODEK DOL
'------------------------
'------------------------
'POMIAR DO WYJ!! PRZEROBIC NA STD
MOVJ C00001 BC00001 VJ=40.00
MOVJ C00002 BC00002 VJ=40.00
'SPOINA_PODLOGA_BRAK_ROZP
MOVJ C00003 BC00003 VJ=20.00 PL=0
MOVL C00004 BC00004 V=166.7 PL=0
REFP 3 C00005 BC00005
CALL JOB:SEARCH-R1
SET P0098 P0006
SFTON P0098
MOVL C00006 BC00006 V=66.7 PL=0
REFP 3 C00007 BC00007
CALL JOB:SEARCH-R1
SET P0098 P0006
SFTON P0098
MOVL C00008 BC00008 V=333.3 PL=0
SFTOF
'W3L
MOVL C00009 BC00009 V=666.7
MOVL C00010 BC00010 V=166.7 PL=0
REFP 3 C00011 BC00011
CALL JOB:SEARCH-R1
SET P0099 P0006
SFTON P0099
MOVL C00012 BC00012 V=166.7 PL=0
REFP 3 C00013 BC00013
CALL JOB:SEARCH-R1
SET P0099 P0006
SFTON P0099
MOVL C00014 BC00014 V=333.3 PL=0
SFTOF
'SPOINA_PODLOGA_BRAK_ROZP
MOVJ C00015 BC00015 VJ=40.00
'W3P
MOVJ C00016 BC00016 VJ=20.00 PL=0
MOVL C00017 BC00017 V=166.7 PL=0
REFP 3 C00018 BC00018
CALL JOB:SEARCH-R1
SET P0100 P0006
SFTON P0100
MOVL C00019 BC00019 V=66.7 PL=0
REFP 3 C00020 BC00020
CALL JOB:SEARCH-R1
SET P0100 P0006
SFTON P0100
MOVL C00021 BC00021 V=333.3 PL=0
SFTOF
'W3L
MOVL C00022 BC00022 V=666.7
MOVL C00023 BC00023 V=166.7 PL=0
REFP 3 C00024 BC00024
CALL JOB:SEARCH-R1
SET P0101 P0006
SFTON P0101
MOVL C00025 BC00025 V=166.7 PL=0
REFP 3 C00026 BC00026
CALL JOB:SEARCH-R1
SET P0101 P0006
SFTON P0101
MOVL C00027 BC00027 V=333.3 PL=0
SFTOF
'W9P
MOVL C00028 BC00028 V=666.7
MOVL C00029 BC00029 V=166.7
REFP 3 C00030 BC00030
CALL JOB:SEARCH-R1
SET P0102 P0006
SFTON P0102
MOVL C00031 BC00031 V=166.7 PL=0
REFP 3 C00032 BC00032
CALL JOB:SEARCH-R1
SET P0102 P0006
SFTON P0102
SFTOF
MOVL C00033 BC00033 V=333.3 PL=0
'W9L
MOVL C00034 BC00034 V=666.7
MOVL C00035 BC00035 V=166.7
REFP 3 C00036 BC00036
CALL JOB:SEARCH-R1
SET P0103 P0006
SFTON P0103
MOVL C00037 BC00037 V=166.7 PL=0
REFP 3 C00038 BC00038
CALL JOB:SEARCH-R1
SET P0103 P0006
SFTON P0103
MOVL C00039 BC00039 V=333.3 PL=0
SFTOF
'PRZEJAZ NAD BELKA
MOVL C00040 BC00040 V=666.7
MOVJ C00041 BC00041 VJ=40.00
MOVJ C00042 BC00042 VJ=40.00
MOVJ C00043 BC00043 VJ=40.00
'W1P
SFTOF
MOVJ C00044 BC00044 VJ=20.00 PL=0
MOVL C00045 BC00045 V=166.7 PL=0
REFP 3 C00046 BC00046
CALL JOB:SEARCH-R1
SET P0104 P0006
SFTON P0104
MOVL C00047 BC00047 V=166.7 PL=0
REFP 3 C00048 BC00048
CALL JOB:SEARCH-R1
SET P0104 P0006
SFTON P0104
MOVL C00049 BC00049 V=333.3 PL=0
SFTOF
'W1L
MOVL C00050 BC00050 V=666.7
MOVL C00051 BC00051 V=166.7 PL=0
REFP 3 C00052 BC00052
CALL JOB:SEARCH-R1
SET P0105 P0006
SFTON P0105
MOVL C00053 BC00053 V=166.7 PL=0
REFP 3 C00054 BC00054
CALL JOB:SEARCH-R1
SET P0105 P0006
SFTON P0105
MOVL C00055 BC00055 V=333.3 PL=0
SFTOF
MOVL C00056 BC00056 V=666.7
'W10P
MOVL C00057 BC00057 V=166.7 PL=0
REFP 3 C00058 BC00058
CALL JOB:SEARCH-R1
SET P0106 P0006
SFTON P0106
MOVL C00059 BC00059 V=166.7 PL=0
REFP 3 C00060 BC00060
CALL JOB:SEARCH-R1
SET P0106 P0006
SFTON P0106
MOVL C00061 BC00061 V=333.3 PL=0
SFTOF
'W10L
MOVL C00062 BC00062 V=333.3
MOVL C00063 BC00063 V=166.7 PL=0
REFP 3 C00064 BC00064
CALL JOB:SEARCH-R1
SET P0107 P0006
SFTON P0107
MOVL C00065 BC00065 V=166.7 PL=0
REFP 3 C00066 BC00066
CALL JOB:SEARCH-R1
SET P0107 P0006
SFTON P0107
MOVL C00067 BC00067 V=333.3 PL=0
SFTOF
MOVL C00068 BC00068 V=333.3
MOVL C00069 BC00069 V=333.3
MOVL C00070 BC00070 V=333.3
MOVL C00071 BC00071 V=833.3
MOVL C00072 BC00072 V=333.3
MOVL C00073 BC00073 V=166.7 PL=0
REFP 3 C00074 BC00074
CALL JOB:SEARCH-R1
SET P0108 P0006
SFTON P0108
MOVL C00075 BC00075 V=166.7 PL=0
REFP 3 C00076 BC00076
CALL JOB:SEARCH-R1
SET P0108 P0006
SFTON P0108
MOVL C00077 BC00077 V=333.3 PL=0
SFTOF
'PRZEJAZD
MOVL C00078 BC00078 V=666.7
MOVL C00079 BC00079 V=166.7 PL=0
REFP 3 C00080 BC00080
CALL JOB:SEARCH-R1
SET P0109 P0006
SFTON P0109
MOVL C00081 BC00081 V=166.7 PL=0
REFP 3 C00082 BC00082
CALL JOB:SEARCH-R1
SET P0109 P0006
SFTON P0109
MOVL C00083 BC00083 V=333.3 PL=0
SFTOF
'PRZEJAZD
'POMIAR DO WYJ!! PRZEROBIC NA STD
'KONIEC
MOVJ C00084 BC00084 VJ=25.00
MOVJ C00085 BC00085 VJ=50.00
'W5L
MOVJ C00086 BC00086 VJ=30.00 PL=0
MOVL C00087 BC00087 V=166.7
REFP 3 C00088 BC00088
CALL JOB:SEARCH-R1
SET P0021 P0006
SFTON P0021
MOVL C00089 BC00089 V=166.7
REFP 3 C00090 BC00090
CALL JOB:SEARCH-R1
SET P0021 P0006
SFTON P0021
SFTOF
MOVL C00091 BC00091 V=166.7
'W6L
MOVJ C00092 BC00092 VJ=20.00 PL=0
MOVL C00093 BC00093 V=166.7
REFP 3 C00094 BC00094
CALL JOB:SEARCH-R1
SET P0022 P0006
SFTON P0022
MOVL C00095 BC00095 V=166.7
REFP 3 C00096 BC00096
CALL JOB:SEARCH-R1
SET P0022 P0006
SFTON P0022
SFTOF
MOVL C00097 BC00097 V=166.7
'W6P
MOVL C00098 BC00098 V=333.3 PL=0
REFP 3 C00099 BC00099
CALL JOB:SEARCH-R1
SET P0023 P0006
SFTON P0023
MOVL C00100 BC00100 V=166.7
REFP 3 C00101 BC00101
CALL JOB:SEARCH-R1
SET P0023 P0006
SFTON P0023
SFTOF
MOVL C00102 BC00102 V=166.7
'W5P
MOVJ C00103 BC00103 VJ=20.00 PL=0
MOVL C00104 BC00104 V=166.7
REFP 3 C00105 BC00105
CALL JOB:SEARCH-R1
SET P0024 P0006
SFTON P0024
MOVL C00106 BC00106 V=166.7
REFP 3 C00107 BC00107
CALL JOB:SEARCH-R1
SET P0024 P0006
SFTON P0024
SFTOF
MOVL C00108 BC00108 V=166.7
'W7A
MOVJ C00109 BC00109 VJ=40.00
MOVJ C00110 BC00110 VJ=40.00
MOVJ C00111 BC00111 VJ=40.00
MOVJ C00112 BC00112 VJ=40.00
MOVJ C00113 BC00113 VJ=40.00
MOVJ C00114 BC00114 VJ=40.00
MOVJ C00115 BC00115 VJ=40.00
MOVJ C00116 BC00116 VJ=40.00
MOVL C00117 BC00117 V=250.0
REFP 3 C00118 BC00118
CALL JOB:SEARCH-R1
SET P0280 P0006
SFTON P0280
MOVL C00119 BC00119 V=166.7
MOVL C00120 BC00120 V=250.0
MOVL C00121 BC00121 V=166.7
REFP 3 C00122 BC00122
CALL JOB:SEARCH-R1
SET P0280 P0006
MOVL C00123 BC00123 V=166.7
SFTOF
MOVL C00124 BC00124 V=333.3
MOVL C00125 BC00125 V=166.7
REFP 3 C00126 BC00126
CALL JOB:SEARCH-R1
SET P0290 P0006
SFTON P0290
MOVL C00127 BC00127 V=166.7
REFP 3 C00128 BC00128
CALL JOB:SEARCH-R1
SET P0290 P0006
MOVL C00129 BC00129 V=166.7
'DOKONCZYC SEARCH
'DOKONCZYC SEARCH
MOVJ C00130 BC00130 VJ=20.00
SFTOF
MOVJ C00131 BC00131 VJ=30.00
MOVJ C00132 BC00132 VJ=40.00
MOVJ C00133 BC00133 VJ=40.00
MOVJ C00134 BC00134 VJ=40.00
MOVJ C00135 BC00135 VJ=40.00
MOVJ C00136 BC00136 VJ=50.00
'W7B
MOVJ C00137 BC00137 VJ=50.00
MOVJ C00138 BC00138 VJ=50.00
MOVJ C00139 BC00139 VJ=30.00
MOVJ C00140 BC00140 VJ=20.00
MOVL C00141 BC00141 V=166.7
REFP 3 C00142 BC00142
CALL JOB:SEARCH-R1
SET P0281 P0006
MOVL C00143 BC00143 V=166.7
SFTON P0281
MOVL C00144 BC00144 V=166.7
MOVL C00145 BC00145 V=166.7
REFP 3 C00146 BC00146
CALL JOB:SEARCH-R1
SET P0281 P0006
MOVJ C00147 BC00147 VJ=15.00
SFTOF
MOVJ C00148 BC00148 VJ=20.00
MOVL C00149 BC00149 V=166.7
REFP 3 C00150 BC00150
CALL JOB:SEARCH-R1
SET P0291 P0006
MOVL C00151 BC00151 V=166.7
MOVL C00152 BC00152 V=166.7
REFP 3 C00153 BC00153
CALL JOB:SEARCH-R1
SET P0291 P0006
MOVL C00154 BC00154 V=166.7
MOVJ C00155 BC00155 VJ=30.00
MOVJ C00156 BC00156 VJ=30.00
MOVJ C00157 BC00157 VJ=50.00
MOVJ C00158 BC00158 VJ=50.00
'------------------------
'------------------------
'PRAWA STRONA PROFIL GORA
'------------------------
'------------------------
MOVJ C00159 BC00159 VJ=50.00
MOVJ C00160 BC00160 VJ=50.00
MOVJ C00161 BC00161 VJ=50.00
MOVJ C00162 BC00162 VJ=20.00
MOVJ C00163 BC00163 VJ=50.00
'------------------------
'W14A L
'------------------------
SFTOF
MOVJ C00164 BC00164 VJ=50.00
'------------------------
'W14A P
'------------------------
SFTOF
MOVJ C00165 BC00165 VJ=50.00
MOVJ C00166 BC00166 VJ=50.00
MOVL C00167 BC00167 V=166.7 PL=0
REFP 3 C00168 BC00168
CALL JOB:SEARCH-R1
SET P0301 P0006
SFTON P0301
MOVL C00169 BC00169 V=166.7 PL=0
REFP 3 C00170 BC00170
CALL JOB:SEARCH-R1
SET P0301 P0006
SFTON P0301
MOVL C00171 BC00171 V=166.7 PL=0
SFTOF
'------------------------
'W19A L
'------------------------
SFTOF
MOVJ C00172 BC00172 VJ=50.00
MOVL C00173 BC00173 V=200.0 PL=0
REFP 3 C00174 BC00174
CALL JOB:SEARCH-R1
SET P0302 P0006
SFTON P0302
MOVL C00175 BC00175 V=166.7 PL=0
REFP 3 C00176 BC00176
CALL JOB:SEARCH-R1
SET P0302 P0006
SFTON P0302
MOVL C00177 BC00177 V=250.0 PL=0
SFTOF
'------------------------
'W19A P
'------------------------
SFTOF
MOVJ C00178 BC00178 VJ=50.00
MOVL C00179 BC00179 V=166.7 PL=0
REFP 3 C00180 BC00180
CALL JOB:SEARCH-R1
SET P0303 P0006
SFTON P0303
MOVL C00181 BC00181 V=166.7 PL=0
REFP 3 C00182 BC00182
CALL JOB:SEARCH-R1
SET P0303 P0006
SFTON P0303
MOVL C00183 BC00183 V=166.7 PL=0
SFTOF
'------------------------
'W13A L
'------------------------
SFTOF
MOVJ C00184 BC00184 VJ=50.00
MOVL C00185 BC00185 V=166.7 PL=0
REFP 3 C00186 BC00186
CALL JOB:SEARCH-R1
SET P0304 P0006
SFTON P0304
MOVL C00187 BC00187 V=166.7 PL=0
REFP 3 C00188 BC00188
CALL JOB:SEARCH-R1
SET P0304 P0006
SFTON P0304
MOVL C00189 BC00189 V=166.7 PL=0
SFTOF
'------------------------
'W13A P
'------------------------
SFTOF
MOVJ C00190 BC00190 VJ=50.00
MOVL C00191 BC00191 V=200.0 PL=0
REFP 3 C00192 BC00192
CALL JOB:SEARCH-R1
SET P0305 P0006
SFTON P0305
MOVL C00193 BC00193 V=166.7 PL=0
REFP 3 C00194 BC00194
CALL JOB:SEARCH-R1
SET P0305 P0006
SFTON P0305
MOVL C00195 BC00195 V=250.0 PL=0
SFTOF
'------------------------
'W18A L
'------------------------
SFTOF
MOVJ C00196 BC00196 VJ=50.00
MOVL C00197 BC00197 V=200.0 PL=0
REFP 3 C00198 BC00198
CALL JOB:SEARCH-R1
SET P0306 P0006
SFTON P0306
MOVL C00199 BC00199 V=166.7 PL=0
REFP 3 C00200 BC00200
CALL JOB:SEARCH-R1
SET P0306 P0006
SFTON P0306
MOVL C00201 BC00201 V=166.7 PL=0
SFTOF
'------------------------
'W18A P
'------------------------
SFTOF
MOVJ C00202 BC00202 VJ=50.00
MOVL C00203 BC00203 V=200.0 PL=0
REFP 3 C00204 BC00204
CALL JOB:SEARCH-R1
SET P0307 P0006
SFTON P0307
MOVL C00205 BC00205 V=166.7 PL=0
REFP 3 C00206 BC00206
CALL JOB:SEARCH-R1
SET P0307 P0006
SFTON P0307
MOVL C00207 BC00207 V=166.7 PL=0
SFTOF
'------------------------
'W15A L
'------------------------
SFTOF
MOVJ C00208 BC00208 VJ=50.00
MOVL C00209 BC00209 V=200.0 PL=0
REFP 3 C00210 BC00210
CALL JOB:SEARCH-R1
SET P0308 P0006
SFTON P0308
MOVL C00211 BC00211 V=166.7 PL=0
REFP 3 C00212 BC00212
CALL JOB:SEARCH-R1
SET P0308 P0006
SFTON P0308
MOVL C00213 BC00213 V=166.7 PL=0
SFTOF
'------------------------
'W15A P
'------------------------
SFTOF
MOVJ C00214 BC00214 VJ=50.00
MOVL C00215 BC00215 V=166.7 PL=0
REFP 3 C00216 BC00216
CALL JOB:SEARCH-R1
SET P0309 P0006
SFTON P0309
MOVL C00217 BC00217 V=166.7 PL=0
REFP 3 C00218 BC00218
CALL JOB:SEARCH-R1
SET P0309 P0006
SFTON P0309
MOVL C00219 BC00219 V=166.7 PL=0
SFTOF
MOVL C00220 BC00220 V=333.3
'------------------------
'W17A L
'------------------------
MOVL C00221 BC00221 V=500.0
SFTOF
MOVJ C00222 BC00222 VJ=20.00
MOVL C00223 BC00223 V=166.7 PL=0
REFP 3 C00224 BC00224
CALL JOB:SEARCH-R1
SET P0310 P0006
SFTON P0310
MOVL C00225 BC00225 V=166.7 PL=0
REFP 3 C00226 BC00226
CALL JOB:SEARCH-R1
SET P0310 P0006
SFTON P0310
MOVL C00227 BC00227 V=166.7 PL=0
SFTOF
'------------------------
'W17A P
'------------------------
SFTOF
MOVL C00228 BC00228 V=416.7
MOVL C00229 BC00229 V=166.7 PL=0
REFP 3 C00230 BC00230
CALL JOB:SEARCH-R1
SET P0311 P0006
SFTON P0311
MOVL C00231 BC00231 V=166.7 PL=0
REFP 3 C00232 BC00232
CALL JOB:SEARCH-R1
SET P0311 P0006
SFTON P0311
MOVL C00233 BC00233 V=166.7 PL=0
SFTOF
MOVJ C00234 BC00234 VJ=10.00
MOVJ C00235 BC00235 VJ=20.00
MOVJ C00236 BC00236 VJ=50.00
MOVJ C00237 BC00237 VJ=50.00
MOVJ C00238 BC00238 VJ=70.00
MOVJ C00239 BC00239 VJ=30.00
MOVJ C00240 BC00240 VJ=30.00
'------------------------
'------------------------
'LEWA STRONA PROFIL GORA
'------------------------
'------------------------
MOVJ C00241 BC00241 VJ=30.00
MOVJ C00242 BC00242 VJ=30.00
MOVJ C00243 BC00243 VJ=30.00
'------------------------
'W17B L
'------------------------
SFTOF
MOVJ C00244 BC00244 VJ=15.00
MOVL C00245 BC00245 V=166.7 PL=0
REFP 3 C00246 BC00246
CALL JOB:SEARCH-R1
SET P0350 P0006
SFTON P0350
MOVL C00247 BC00247 V=166.7 PL=0
REFP 3 C00248 BC00248
CALL JOB:SEARCH-R1
SET P0350 P0006
SFTON P0350
MOVL C00249 BC00249 V=166.7 PL=0
SFTOF
'------------------------
'W17B P
'------------------------
SFTOF
MOVL C00250 BC00250 V=333.3
MOVL C00251 BC00251 V=166.7 PL=0
REFP 3 C00252 BC00252
CALL JOB:SEARCH-R1
SET P0351 P0006
SFTON P0351
MOVL C00253 BC00253 V=166.7 PL=0
REFP 3 C00254 BC00254
CALL JOB:SEARCH-R1
SET P0351 P0006
SFTON P0351
MOVL C00255 BC00255 V=166.7 PL=0
SFTOF
'POPRAWID DOJAZD
'------------------------
'W15B L
'------------------------
SFTOF
MOVJ C00256 BC00256 VJ=10.00
MOVL C00257 BC00257 V=166.7 PL=0
REFP 3 C00258 BC00258
CALL JOB:SEARCH-R1
SET P0352 P0006
SFTON P0352
MOVL C00259 BC00259 V=166.7 PL=0
REFP 3 C00260 BC00260
CALL JOB:SEARCH-R1
SET P0352 P0006
SFTON P0352
MOVL C00261 BC00261 V=166.7 PL=0
SFTOF
'------------------------
'W15B P
'------------------------
SFTOF
MOVJ C00262 BC00262 VJ=20.00
MOVL C00263 BC00263 V=166.7 PL=0
REFP 3 C00264 BC00264
CALL JOB:SEARCH-R1
SET P0353 P0006
SFTON P0353
MOVL C00265 BC00265 V=166.7 PL=0
REFP 3 C00266 BC00266
CALL JOB:SEARCH-R1
SET P0353 P0006
SFTON P0353
MOVL C00267 BC00267 V=166.7 PL=0
SFTOF
'------------------------
'W18B L
'------------------------
SFTOF
MOVJ C00268 BC00268 VJ=50.00
MOVL C00269 BC00269 V=166.7 PL=0
REFP 3 C00270 BC00270
CALL JOB:SEARCH-R1
SET P0354 P0006
SFTON P0354
MOVL C00271 BC00271 V=166.7 PL=0
REFP 3 C00272 BC00272
CALL JOB:SEARCH-R1
SET P0354 P0006
SFTON P0354
MOVL C00273 BC00273 V=166.7 PL=0
SFTOF
'------------------------
'W18B P
'------------------------
SFTOF
MOVJ C00274 BC00274 VJ=50.00
MOVL C00275 BC00275 V=166.7 PL=0
REFP 3 C00276 BC00276
CALL JOB:SEARCH-R1
SET P0355 P0006
SFTON P0355
MOVL C00277 BC00277 V=166.7 PL=0
REFP 3 C00278 BC00278
CALL JOB:SEARCH-R1
SET P0355 P0006
SFTON P0355
MOVL C00279 BC00279 V=166.7 PL=0
SFTOF
'------------------------
'W13B L
'------------------------
SFTOF
MOVJ C00280 BC00280 VJ=50.00
MOVL C00281 BC00281 V=166.7 PL=0
REFP 3 C00282 BC00282
CALL JOB:SEARCH-R1
SET P0356 P0006
SFTON P0356
MOVL C00283 BC00283 V=166.7 PL=0
REFP 3 C00284 BC00284
CALL JOB:SEARCH-R1
SET P0356 P0006
SFTON P0356
MOVL C00285 BC00285 V=166.7 PL=0
SFTOF
'------------------------
'W13B P
'------------------------
SFTOF
MOVJ C00286 BC00286 VJ=50.00
MOVL C00287 BC00287 V=166.7 PL=0
REFP 3 C00288 BC00288
CALL JOB:SEARCH-R1
SET P0357 P0006
SFTON P0357
MOVL C00289 BC00289 V=166.7 PL=0
REFP 3 C00290 BC00290
CALL JOB:SEARCH-R1
SET P0357 P0006
SFTON P0357
MOVL C00291 BC00291 V=166.7 PL=0
SFTOF
'------------------------
'W19B L
'------------------------
SFTOF
MOVJ C00292 BC00292 VJ=50.00
MOVL C00293 BC00293 V=166.7 PL=0
REFP 3 C00294 BC00294
CALL JOB:SEARCH-R1
SET P0358 P0006
SFTON P0358
MOVL C00295 BC00295 V=166.7 PL=0
REFP 3 C00296 BC00296
CALL JOB:SEARCH-R1
SET P0358 P0006
SFTON P0358
MOVL C00297 BC00297 V=166.7 PL=0
SFTOF
'------------------------
'W19B P
'------------------------
SFTOF
MOVJ C00298 BC00298 VJ=50.00
MOVL C00299 BC00299 V=166.7 PL=0
REFP 3 C00300 BC00300
CALL JOB:SEARCH-R1
SET P0359 P0006
SFTON P0359
MOVL C00301 BC00301 V=166.7 PL=0
REFP 3 C00302 BC00302
CALL JOB:SEARCH-R1
SET P0359 P0006
SFTON P0359
MOVL C00303 BC00303 V=166.7 PL=0
SFTOF
'------------------------
'W14B L
'------------------------
SFTOF
MOVJ C00304 BC00304 VJ=50.00
MOVL C00305 BC00305 V=166.7 PL=0
REFP 3 C00306 BC00306
CALL JOB:SEARCH-R1
SET P0360 P0006
SFTON P0360
MOVL C00307 BC00307 V=166.7 PL=0
REFP 3 C00308 BC00308
CALL JOB:SEARCH-R1
SET P0360 P0006
SFTON P0360
MOVL C00309 BC00309 V=166.7 PL=0
SFTOF
'------------------------
'W14B P
'------------------------
SFTOF
SFTOF
MOVJ C00310 BC00310 VJ=50.00
MOVJ C00311 BC00311 VJ=50.00
MOVJ C00312 BC00312 VJ=50.00
'WELD
'WELD
'WELD
MOVJ C00313 BC00313 VJ=10.00
'**********************
'**********************
'POCZATEK SPAWANIA DOL
'**********************
'**********************
''
'**********************
'W1
'**********************
MOVJ C00314 BC00314 VJ=50.00
MOVJ C00315 BC00315 VJ=40.00
MOVL C00316 BC00316 V=166.7
SFTON P0105
MOVL C00317 BC00317 V=166.7 PL=0
MACRO1 MJ#(0) ARGF24
ARCON
SFTON P0104
MOVL C00318 BC00318 V=11.3
MOVL C00319 BC00319 V=11.3
ARCOF
SFTOF
MOVL C00320 BC00320 V=333.3
MOVJ C00321 BC00321 VJ=20.00
MOVJ C00322 BC00322 VJ=30.00
MOVJ C00323 BC00323 VJ=50.00
MOVJ C00324 BC00324 VJ=40.00
MOVJ C00325 BC00325 VJ=20.00
'**********************
'W2
'**********************
MOVL C00326 BC00326 V=166.7
SFTON P0109
MOVL C00327 BC00327 V=333.3
ARCON
SFTON P0108
MOVL C00328 BC00328 V=10.8
ARCOF
SFTOF
MOVL C00329 BC00329 V=333.3
MOVJ C00330 BC00330 VJ=40.00
MOVJ C00331 BC00331 VJ=70.00
MOVJ C00332 BC00332 VJ=20.00
MOVL C00333 BC00333 V=666.7
'**********************
'W3
'**********************
SFTON P0101
MOVL C00334 BC00334 V=166.7 PL=0
ARCON
SFTON P0100
MOVL C00335 BC00335 V=11.7
ARCOF
MOVL C00336 BC00336 V=166.7
SFTOF
MOVJ C00337 BC00337 VJ=30.00
MOVJ C00338 BC00338 VJ=30.00
MOVJ C00339 BC00339 VJ=50.00
MOVJ C00340 BC00340 VJ=30.00
MOVJ C00341 BC00341 VJ=40.00
'**********************
'W5
'**********************
MOVJ C00342 BC00342 VJ=50.00
MOVJ C00343 BC00343 VJ=25.00
MOVJ C00344 BC00344 VJ=30.00
'**********************
'W5
MOVL C00345 BC00345 V=333.3
'**********************
MACRO1 MJ#(0) ARGF9
SFTON P0024
MOVL C00346 BC00346 V=166.7 PL=0
ARCON
WVON WEV#(2)
SFTON P0021
MOVL C00347 BC00347 V=10.8
ARCOF
WVOF
SFTOF
MOVJ C00348 BC00348 VJ=20.00
MOVJ C00349 BC00349 VJ=20.00
'**********************
'W6
'**********************
MACRO1 MJ#(0) ARGF9
SFTON P0023
MOVL C00350 BC00350 V=250.0
ARCON
WVON WEV#(2)
SFTON P0022
MOVL C00351 BC00351 V=10.8
ARCOF
WVOF
SFTOF
MOVJ C00352 BC00352 VJ=10.00
MOVJ C00353 BC00353 VJ=30.00
MOVJ C00354 BC00354 VJ=40.00
MOVJ C00355 BC00355 VJ=40.00
MOVJ C00356 BC00356 VJ=40.00
MOVJ C00357 BC00357 VJ=40.00
MOVJ C00358 BC00358 VJ=20.00
MOVJ C00359 BC00359 VJ=10.00
MOVJ C00360 BC00360 VJ=20.00
MOVL C00361 BC00361 V=166.7
MACRO1 MJ#(0) ARGF14
MOVL C00362 BC00362 V=166.7
SFTON P0280
MOVL C00363 BC00363 V=166.7 PL=0
ARCON ASF#(22)
MOVL C00364 BC00364 V=9.2
MOVL C00365 BC00365 V=9.2
SFTON P0290
MOVL C00366 BC00366 V=9.2
MOVL C00367 BC00367 V=9.2
ARCOF
SFTOF
MOVL C00368 BC00368 V=250.0
MOVL C00369 BC00369 V=416.7
MOVJ C00370 BC00370 VJ=30.00
MOVJ C00371 BC00371 VJ=30.00
MOVJ C00372 BC00372 VJ=30.00
MOVJ C00373 BC00373 VJ=30.00
MOVJ C00374 BC00374 VJ=30.00
'7b
MOVL C00375 BC00375 V=333.3
MOVL C00376 BC00376 V=333.3
SFTON P0281
MOVL C00377 BC00377 V=166.7 PL=0
ARCON ASF#(22)
MOVL C00378 BC00378 V=9.2
MOVL C00379 BC00379 V=9.2
SFTON P0291
MOVL C00380 BC00380 V=9.2
MOVL C00381 BC00381 V=9.2
MOVL C00382 BC00382 V=9.2
ARCOF
SFTOF
'TUTAJ DODAC 7
'TUTAJ DODAC 7
'TUTAJ DODAC 7
MOVL C00383 BC00383 V=333.3
MOVL C00384 BC00384 V=333.3
MOVL C00385 BC00385 V=333.3
MOVJ C00386 BC00386 VJ=20.00
MOVJ C00387 BC00387 VJ=30.00
MOVJ C00388 BC00388 VJ=50.00
MOVJ C00389 BC00389 VJ=50.00
MOVJ C00390 BC00390 VJ=40.00
'**********************
'W9
'**********************
MACRO1 MJ#(0) ARGF24
MOVL C00391 BC00391 V=166.7
SFTON P0102
MOVL C00392 BC00392 V=166.7 PL=0
ARCON
SFTON P0103
MOVL C00393 BC00393 V=11.3
ARCOF
SFTOF
MOVL C00394 BC00394 V=333.3
'**********************
'SPOINA_PODLOGA_BRAK_ROZP
'**********************
MOVL C00395 BC00395 V=333.3
SFTON P0099
MOVL C00396 BC00396 V=166.7
ARCON
SFTON P0098
MOVL C00397 BC00397 V=11.7
ARCOF
MOVL C00398 BC00398 V=166.7
SFTOF
'SPOINA_PODLOGA_BRAK_ROZP
MOVJ C00399 BC00399 VJ=25.00
MOVJ C00400 BC00400 VJ=40.00
MOVJ C00401 BC00401 VJ=70.00
MOVJ C00402 BC00402 VJ=50.00
MOVJ C00403 BC00403 VJ=20.00
'**********************
'W10
'**********************
MOVL C00404 BC00404 V=333.3
SFTON P0106
MOVL C00405 BC00405 V=166.7 PL=0
ARCON
SFTON P0107
MOVL C00406 BC00406 V=11.3
ARCOF
SFTOF
MOVL C00407 BC00407 V=333.3
MOVJ C00408 BC00408 VJ=50.00
'**********************
'**********************
'POCZATEK SPAWANIA BOKI
'**********************
'**********************
MOVJ C00409 BC00409 VJ=50.00
MOVJ C00410 BC00410 VJ=50.00
'**********************
'W13A
'**********************
SFTON P0305
MOVL C00411 BC00411 V=250.0 PL=0
SFTOF
MACRO1 MJ#(0) ARGF10
ARCON
SFTON P0304
MOVL C00412 BC00412 V=10.8
ARCOF
SFTOF
MOVL C00413 BC00413 V=250.0
'W13B
MOVJ C00414 BC00414 VJ=30.00
MOVJ C00415 BC00415 VJ=50.00
MOVL C00416 BC00416 V=500.0
'**********************
'W13B
'**********************
SFTON P0356
MOVL C00417 BC00417 V=166.7 PL=0
SFTOF
ARCON
SFTON P0357
MOVL C00418 BC00418 V=10.8
ARCOF
SFTOF
MOVL C00419 BC00419 V=250.0
MOVJ C00420 BC00420 VJ=30.00
MOVJ C00421 BC00421 VJ=40.00
MOVJ C00422 BC00422 VJ=30.00
MOVJ C00423 BC00423 VJ=30.00
'**********************
'W14A
'**********************
MOVL C00424 BC00424 V=250.0
SFTON P0301
MOVL C00425 BC00425 V=133.3 PL=0
SFTOF
ARCON
SFTON P0301
MOVL C00426 BC00426 V=10.8
ARCOF
SFTOF
MOVL C00427 BC00427 V=150.0
MOVJ C00428 BC00428 VJ=40.00
MOVJ C00429 BC00429 VJ=30.00
MOVJ C00430 BC00430 VJ=30.00
MOVJ C00431 BC00431 VJ=30.00
MOVJ C00432 BC00432 VJ=30.00
'**********************
'W14B
'**********************
SFTON P0360
MOVL C00433 BC00433 V=333.3
MOVL C00434 BC00434 V=166.7 PL=0
ARCON
MOVL C00435 BC00435 V=10.8
ARCOF
SFTOF
MOVL C00436 BC00436 V=250.0
MOVJ C00437 BC00437 VJ=40.00
MOVJ C00438 BC00438 VJ=40.00
MOVJ C00439 BC00439 VJ=30.00
MOVJ C00440 BC00440 VJ=40.00
MOVJ C00441 BC00441 VJ=30.00
MOVJ C00442 BC00442 VJ=30.00
MOVJ C00443 BC00443 VJ=30.00
MOVJ C00444 BC00444 VJ=30.00
MOVJ C00445 BC00445 VJ=30.00
'**********************
'W15A
'**********************
SFTON P0309
MOVL C00446 BC00446 V=166.7
MOVL C00447 BC00447 V=166.7 PL=0
SFTOF
ARCON
SFTON P0308
MOVL C00448 BC00448 V=10.8
ARCOF
SFTOF
MOVL C00449 BC00449 V=150.0
MOVJ C00450 BC00450 VJ=30.00
MOVJ C00451 BC00451 VJ=50.00
MOVJ C00452 BC00452 VJ=50.00
MOVJ C00453 BC00453 VJ=50.00
MOVJ C00454 BC00454 VJ=50.00
MOVJ C00455 BC00455 VJ=50.00
'**********************
'W15B
'**********************
SFTON P0352
MOVL C00456 BC00456 V=250.0
MOVL C00457 BC00457 V=83.3 PL=0
SFTOF
ARCON
SFTON P0353
MOVL C00458 BC00458 V=10.8
ARCOF
MOVL C00459 BC00459 V=66.7
SFTOF
MOVJ C00460 BC00460 VJ=40.00
MOVJ C00461 BC00461 VJ=50.00
MOVJ C00462 BC00462 VJ=50.00
'BRAK W TEJ DLUGOSCI
'**********************
'W16A
'**********************
'**********************
'W16B
'**********************
'BRAK W TEJ DLUGOSCI
'**********************
'W17A
'**********************
MOVJ C00463 BC00463 VJ=50.00
MOVJ C00464 BC00464 VJ=50.00
'**********************
'W17A
'**********************
SFTON P0310
MOVL C00465 BC00465 V=333.3
MOVL C00466 BC00466 V=166.7 PL=0
SFTOF
ARCON
SFTON P0311
MOVL C00467 BC00467 V=10.8
ARCOF
SFTOF
MOVL C00468 BC00468 V=333.3
MOVJ C00469 BC00469 VJ=30.00
MOVJ C00470 BC00470 VJ=30.00
MOVJ C00471 BC00471 VJ=50.00
MOVJ C00472 BC00472 VJ=50.00
MOVJ C00473 BC00473 VJ=50.00
MOVJ C00474 BC00474 VJ=50.00
MOVJ C00475 BC00475 VJ=50.00
MOVJ C00476 BC00476 VJ=30.00
MOVJ C00477 BC00477 VJ=30.00
'**********************
'W17B
'**********************
SFTON P0351
MOVL C00478 BC00478 V=166.7
MOVL C00479 BC00479 V=166.7 PL=0
SFTOF
ARCON
SFTON P0350
MOVL C00480 BC00480 V=10.8
ARCOF
SFTOF
MOVL C00481 BC00481 V=250.0
MOVJ C00482 BC00482 VJ=30.00
MOVJ C00483 BC00483 VJ=30.00
MOVJ C00484 BC00484 VJ=30.00
MOVJ C00485 BC00485 VJ=30.00
MOVJ C00486 BC00486 VJ=40.00
'**********************
'W18A
'**********************
SFTON P0306
MOVL C00487 BC00487 V=333.3
MOVL C00488 BC00488 V=166.7 PL=0
SFTOF
ARCON
SFTON P0307
MOVL C00489 BC00489 V=10.8
ARCOF
SFTOF
MOVL C00490 BC00490 V=250.0
MOVJ C00491 BC00491 VJ=30.00
MOVJ C00492 BC00492 VJ=30.00
MOVJ C00493 BC00493 VJ=50.00
MOVJ C00494 BC00494 VJ=50.00
MOVJ C00495 BC00495 VJ=50.00
'**********************
'W18B
'**********************
SFTON P0355
MOVL C00496 BC00496 V=166.7
MOVL C00497 BC00497 V=166.7 PL=0
SFTOF
ARCON
SFTON P0354
MOVL C00498 BC00498 V=10.8
ARCOF
MOVL C00499 BC00499 V=250.0
SFTOF
MOVJ C00500 BC00500 VJ=30.00
MOVJ C00501 BC00501 VJ=30.00
MOVJ C00502 BC00502 VJ=40.00
MOVJ C00503 BC00503 VJ=50.00
MOVJ C00504 BC00504 VJ=30.00
'**********************
'W19A
'**********************
MOVL C00505 BC00505 V=166.7
SFTON P0303
MOVL C00506 BC00506 V=166.7 PL=0
SFTOF
ARCON
SFTON P0302
MOVL C00507 BC00507 V=10.8
ARCOF
SFTOF
MOVL C00508 BC00508 V=150.0
MOVJ C00509 BC00509 VJ=30.00
MOVJ C00510 BC00510 VJ=50.00
MOVJ C00511 BC00511 VJ=50.00
'**********************
'W19B
'**********************
SFTON P0358
MOVL C00512 BC00512 V=500.0
MOVL C00513 BC00513 V=166.7 PL=0
SFTOF
ARCON
SFTON P0359
MOVL C00514 BC00514 V=10.8
ARCOF
SFTOF
MOVL C00515 BC00515 V=250.0
MOVJ C00516 BC00516 VJ=40.00
MOVJ C00517 BC00517 VJ=50.00
CALL JOB:MOVE_OUT_OF_TUNNEL
END
